TYPE (* logiBUS_DO Struct *)
  (* Version 1.0, 2025-07-21, Franz Höpfinger, initial API and implementation and/or initial documentation *)
  PACKAGE logiBUS::io::DQ;
  logiBUS_DO_S : STRUCT
    Pin : USINT := 255;
  END_STRUCT;
END_TYPE
